PROGRAM MAIN
VAR
	stGlobalStatus				: ST_GlobalStatus;
END_VAR

stGlobalStatus.nDummy := stGlobalStatus.nDummy + 1;

END_PROGRAM

(* stored: Version 1.1.0.1, ProductVersion 3.1.4024.12
   POU MAIN: Id {158c46bb-c09e-4b61-ae02-fb8da9009f60}, SpecialFunc None *)
